# EPICS substitutions: apps/caenHvApp/Db/seq/hvOnOff.substitutions
file "db/hvOnOff-6sec-1det.db" {
    pattern { DET ONOFF }
    { ECAL ON }
    { ECAL OFF }
    { PCAL ON }
    { PCAL OFF }
    { FTOF ON }
    { FTOF OFF }
    { LTCC ON }
    { LTCC OFF }
    { HTCC ON }
    { HTCC OFF }
}
